RoboDK station: RBT23ME030_ROSHANI.rdk

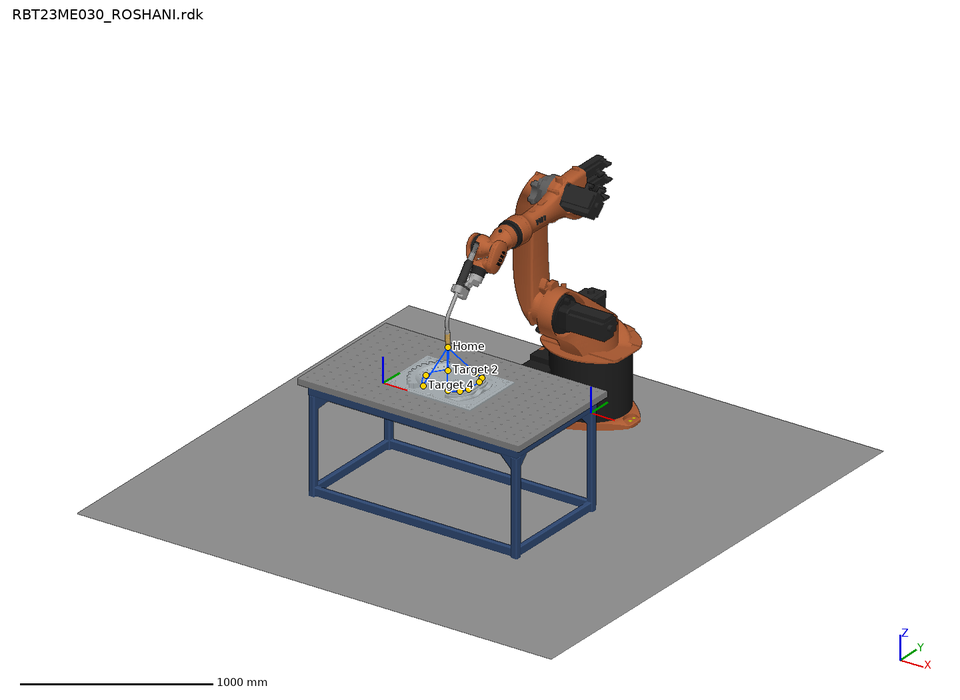
[picture v0: the station drawn from its stored meshes, robots at their saved joint values, targets as dots, program paths as lines]
Station RBT23ME030_ROSHANI (saved by RoboDK 5.9.2). Poses are relative to the parent item; angles as X-Y-Z fixed-axis rotations.
Station parameters (name, value as stored): IO_5, 0
  - frame KUKA KR 16 3 Base at (0, 1000, 0) mm
    - robot KUKA KR 16 3: 6 axes, payload 16 kg, reach 1611 mm, repeatability 0.05 mm, weight 235 kg
        modified DH rows (alpha deg, a mm, theta deg, d mm): 0, 0, 0, 675; -90, 260, 0, 0; 0, 680, -90, 0; -90, -35, 0, 670; 90, 0, 0, 0; -90, 0, 180, 158
        joint limits [-185, -155, -130, -350, -130, -350] to [185, 35, 154, 350, 130, 350]; home [0, -90, 90, 0, 0, 0]; saved at [90, -89.97, 90.017, 0, 49.953, 0]
      - tool Abicor Binzel 45deg Welding Gun, TCP at (0, 0, 400) mm, rotated rx 0 ry 45 rz 0 deg, size 179.1 x 69.8 x 552.4 mm
  - object Table 1400x800x800mm at (-340, -280, 680) mm, size 1420 x 820 x 800 mm, geometry from Table-1400x800x800mm.sld
  - object Floor at (0, 0, 0) mm, size 3000 x 3000 x 0 mm, geometry from Floor.sld
  - frame Reference Frame at (-270, -490, 690) mm
    - object RoboDK Test Plate 550x400mm at (0, 0, 0) mm, size 550 x 400 x 43 mm, geometry from RoboDK-Test-Plate-550x400mm.sld
    - target Home (Cartesian target) at (270, 201.33, 202.55) mm, rotated rx 180 ry -5 rz 90 deg; joints [90, -90, 90, 0, 50, 0] of KUKA KR 16 3
    - target Target 2 (Cartesian target) at (191, 311.33, 2.55) mm, rotated rx 180 ry -5 rz 90 deg; joints [95.503, -95.553, 112.776, -6.485, 33.076, 9.662] of KUKA KR 16 3
    - target Target 3 (Cartesian target) at (131, 201.33, 2.55) mm, rotated rx 180 ry -5 rz 90 deg; joints [98.501, -85.682, 103.019, -9.947, 33.371, 14.864] of KUKA KR 16 3
    - target Target 4 (Cartesian target) at (191, 91.33, 2.55) mm, rotated rx 180 ry -5 rz 90 deg; joints [94.344, -77.371, 93.391, -4.974, 34.161, 7.449] of KUKA KR 16 3
    - target Target 9 (Cartesian target) at (270, 201, 202) mm, rotated rx 180 ry -5 rz 90 deg; joints [90, -89.97, 90.017, 0, 49.953, 0] of KUKA KR 16 3
    - target Target 5 (Cartesian target) at (358, 326, 28) mm, rotated rx 180 ry -5 rz 90 deg; joints [83.764, -97.532, 112.215, 6.876, 35.68, -10.379] of KUKA KR 16 3
    - target Target 11 (Cartesian target) at (415, 300, 28) mm, rotated rx -180 ry -5 rz 90 deg; joints [80.106, -94.57, 109.585, 10.858, 35.897, -16.442] of KUKA KR 16 3
    - target Target 6 (Cartesian target) at (435, 250, 28) mm, rotated rx 180 ry -5 rz 90 deg; joints [79.396, -90.06, 105.269, 11.655, 35.841, -17.654] of KUKA KR 16 3
    - target Target 7 (Cartesian target) at (435, 150, 28) mm, rotated rx 180 ry -5 rz 90 deg; joints [80.456, -81.921, 96.524, 10.387, 36.239, -15.749] of KUKA KR 16 3
    - target Target 12 (Cartesian target) at (415, 100, 28) mm, rotated rx 180 ry -5 rz 90 deg; joints [81.997, -78.158, 92.072, 8.618, 36.674, -13.078] of KUKA KR 16 3
    - target Target 8 (Cartesian target) at (358, 73, 28) mm, rotated rx 180 ry -5 rz 90 deg; joints [85.247, -76.499, 90.027, 5.116, 36.679, -7.751] of KUKA KR 16 3
    - target Target 10 (Cartesian target) at (270, 201, 202) mm, rotated rx -180 ry -5 rz 90 deg; joints [90, -89.97, 90.017, 0, 49.953, 0] of KUKA KR 16 3
  - program Prog1 (17 instructions, listed below)
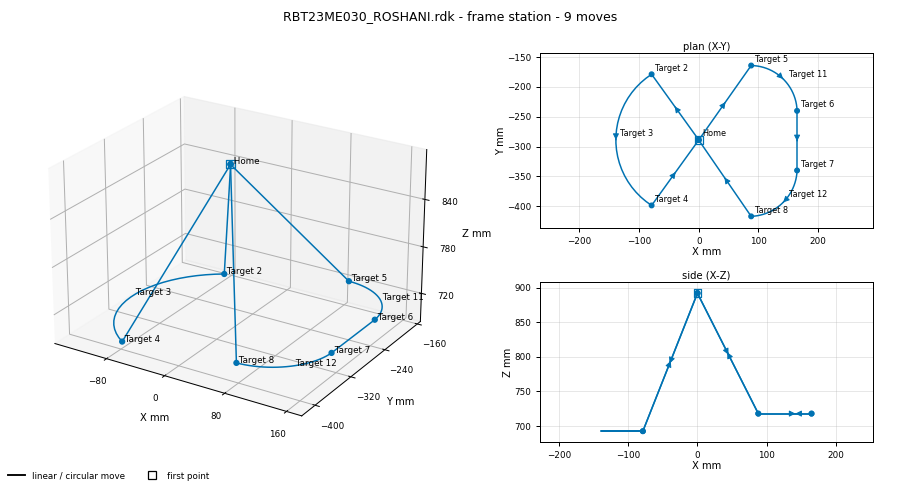
[picture p0: tool path of RBT23ME030_ROSHANI.rdk in frame station, 9 of 9 moves have a stored position in this frame; points joined in program order, loops and branches not executed]

--- program Prog1 (robot KUKA KR 16 3) ---
  Set Ref.: Reference Frame
  Set Tool: Abicor Binzel 45deg Welding Gun
  MoveL (Home)
  MoveL (Target 2)
  Set IO_5=1
  MoveC (Target 3, Target 4)
  Set IO_5=0
  MoveL (Target 9)
  MoveL (Target 5)
  Set IO_5=1
  MoveC (Target 11, Target 6)
  MoveL (Target 7)
  MoveC (Target 12, Target 8)
  Set IO_5=0
  MoveL (Target 10)
  Set speed (10.0 mm/s)
  Set speed (100.0 mm/s)
